{attribute 'GeneratedUsingTerminal: EPP2817-0008-0016'}
{attribute addProperty BoxType "EPP2817-0008-0016"}
{attribute addProperty Id "DIG_Diag_Inputs_Channel_1AT %I*DIG_Diag_Inputs_Channel_584303BF8DIG_Diag_Inputs_Channel_2AT %I*DIG_Diag_Inputs_Channel_584303BF8DIG_Diag_Inputs_Channel_3AT %I*DIG_Diag_Inputs_Channel_584303BF8DIG_Inputs_DeviceAT %I*DIG_Inputs_Device_27CCC8668DIG_Output_Channel_1AT %Q*DIG_Output_Channel_28AC1A9E8DIG_Output_Channel_2AT %Q*DIG_Output_Channel_28AC1A9E8DIG_Output_Channel_3AT %Q*DIG_Output_Channel_28AC1A9E8DIG_Outputs_DeviceAT %Q*DIG_Outputs_Device_36A5EF172WcStateAT %I*WcState_9091E0EB2InfoDataAT %I*InfoData_94A18F5E2"}
{attribute addProperty CRC "3667233126"}
{attribute addProperty Size "62"}
TYPE EPP2817_DA958966 EXTENDS EtcSlaveTerminalBase_947E5A46 :
STRUCT
	{attribute addProperty Name "DIG_Diag_Inputs_Channel_1"}
	DIG_Diag_Inputs_Channel_1 : DIG_Diag_Inputs_Channel_584303BF;
	{attribute addProperty Name "DIG_Diag_Inputs_Channel_2"}
	DIG_Diag_Inputs_Channel_2 : DIG_Diag_Inputs_Channel_584303BF;
	{attribute addProperty Name "DIG_Diag_Inputs_Channel_3"}
	DIG_Diag_Inputs_Channel_3 : DIG_Diag_Inputs_Channel_584303BF;
	{attribute addProperty Name "DIG_Inputs_Device"}
	DIG_Inputs_Device : DIG_Inputs_Device_27CCC866;
	{attribute addProperty Name "DIG_Output_Channel_1"}
	DIG_Output_Channel_1 : DIG_Output_Channel_28AC1A9E;
	{attribute addProperty Name "DIG_Output_Channel_2"}
	DIG_Output_Channel_2 : DIG_Output_Channel_28AC1A9E;
	{attribute addProperty Name "DIG_Output_Channel_3"}
	DIG_Output_Channel_3 : DIG_Output_Channel_28AC1A9E;
	{attribute addProperty Name "DIG_Outputs_Device"}
	DIG_Outputs_Device : DIG_Outputs_Device_36A5EF17;
	{attribute addProperty Name "WcState"}
	WcState : WcState_9091E0EB;
	{attribute addProperty Name "InfoData"}
	InfoData : InfoData_94A18F5E;
END_STRUCT
END_TYPE

(* stored: Version 1.2.0.0, ProductVersion 3.1.4024.9
   DUT EPP2817_DA958966: Id {eb53b3b6-493b-4989-a0a7-2be1e41cb3d8} *)
